ABB RobotStudio station: Project4.rsstnx

Station Project4 (saved by RobotStudio 23.2.10395.0)
Controller IRB140_6_81
  mechanical unit ROB_1: IRB140_6_81_C_03, 6 joints, base frame (0, 0, 0) mm
Layout (positions relative to the parent item):
  - IRB140_6_81_C_03 [mechanism, from %ABB.RobotStudio.Models.IRB140%\IRB140_6_81_C_G_03.rslib] at (0, 0, 0) mm; joint values [0.7528, 0.4246, 0.2198, -0.8632, 0.587, 1.4078] (rad or m)
  - Cubo_2 [part] at (500, 400, 0) mm, rotated rx 90 ry 0 rz 0 deg, size 180 x 200 x 180 mm
  - MyNewTool [mechanism] at (421.04, 356.95, 400.53) mm, rotated rx 180 ry 38 rz 180 deg
      TCP CualquierCosa at (131.19, 0, 127.78) mm, rotated rx 0 ry 75 rz 0 deg
      links: BaseMarcador
  - MyTool [mechanism, from Training Objects\myTool.rslib] at (421.04, 356.95, 400.53) mm, rotated rx 180 ry 38 rz 180 deg
Attachment: MyNewTool is attached to IRB140_6_81_C_03 / Link6
Attachment: MyTool is attached to IRB140_6_81_C_03 / Link6
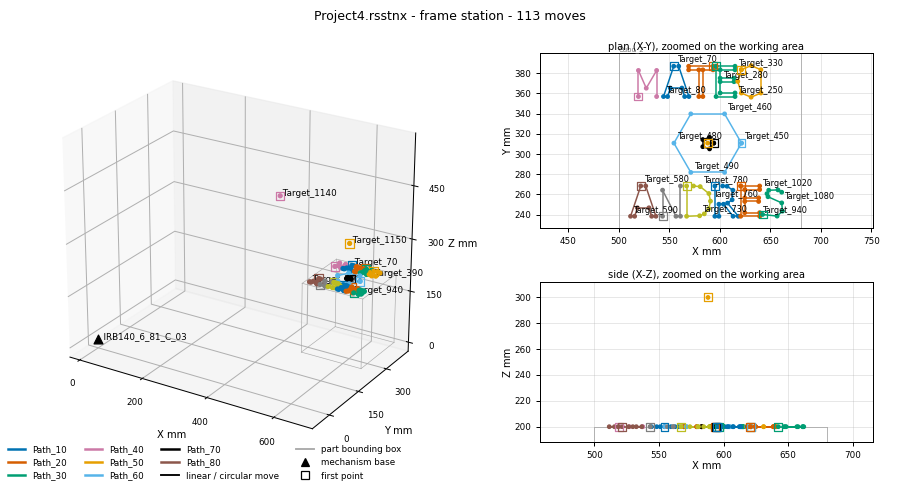
[picture p0: tool path of Project4.rsstnx in frame station, 113 of 113 moves have a stored position in this frame; points joined in program order, loops and branches not executed]
Targets, tools, work objects and paths stored in the station, written as RAPID:
! task T_ROB1
MODULE Module1
  PERS wobjdata Workobject_8:=[FALSE,TRUE,"",[[150,100,0],[1,0,0,0]],[[351.920963746,301.866615458,180],[0,0.710877818,0.703315525,0]]];
  CONST robtarget Target_10:=[[-44.732003119,17.911406594,-20],[0.703315525,0,0,-0.710877818],[0,0,0,0],[9E+09,9E+09,9E+09,9E+09,9E+09,9E+09]];
  CONST robtarget Target_20:=[[-18.89069334,17.635029753,-20],[0.703315525,0,0,-0.710877818],[0,0,0,0],[9E+09,9E+09,9E+09,9E+09,9E+09,9E+09]];
  CONST robtarget Target_30:=[[-36.383734505,25.577831517,-20],[0.703315525,0,0,-0.710877818],[0,0,0,0],[9E+09,9E+09,9E+09,9E+09,9E+09,9E+09]];
  CONST robtarget Target_40:=[[-18.698035542,35.64858624,-20],[0.703315525,0,0,-0.710877818],[0,0,0,0],[9E+09,9E+09,9E+09,9E+09,9E+09,9E+09]];
  CONST robtarget Target_50:=[[-44.539345321,35.924963081,-20],[0.703315525,0,0,-0.710877818],[0,0,0,0],[9E+09,9E+09,9E+09,9E+09,9E+09,9E+09]];
  CONST robtarget Target_60:=[[-14.355335815,52.933587211,-20],[0.703315525,0,0,-0.710877818],[0,0,0,0],[9E+09,9E+09,9E+09,9E+09,9E+09,9E+09]];
  CONST robtarget Target_70:=[[-14.359843041,52.548052351,-20],[0.703315525,0,0,-0.710877818],[0,0,0,0],[9E+09,9E+09,9E+09,9E+09,9E+09,9E+09]];
  CONST robtarget Target_80:=[[-44.466286156,42.756014866,-20],[0.703315525,0,0,-0.710877818],[0,0,0,0],[9E+09,9E+09,9E+09,9E+09,9E+09,9E+09]];
  CONST robtarget Target_90:=[[-44.423126649,46.791440476,-20],[0.703315525,0,0,-0.710877818],[0,0,0,0],[9E+09,9E+09,9E+09,9E+09,9E+09,9E+09]];
  CONST robtarget Target_100:=[[-36.007128456,49.424438298,-20],[0.703315525,0,0,-0.710877818],[0,0,0,0],[9E+09,9E+09,9E+09,9E+09,9E+09,9E+09]];
  CONST robtarget Target_110:=[[-35.884669856,60.874350721,-20],[0.703315525,0,0,-0.710877818],[0,0,0,0],[9E+09,9E+09,9E+09,9E+09,9E+09,9E+09]];
  CONST robtarget Target_120:=[[-44.242428715,63.686746492,-20],[0.703315525,0,0,-0.710877818],[0,0,0,0],[9E+09,9E+09,9E+09,9E+09,9E+09,9E+09]];
  CONST robtarget Target_130:=[[-44.197449229,67.892340652,-20],[0.703315525,0,0,-0.710877818],[0,0,0,0],[9E+09,9E+09,9E+09,9E+09,9E+09,9E+09]];
  CONST robtarget Target_140:=[[-14.307323641,57.458630502,-20],[0.703315525,0,0,-0.710877818],[0,0,0,0],[9E+09,9E+09,9E+09,9E+09,9E+09,9E+09]];
  CONST robtarget Target_150:=[[-13.943587799,91.468030671,-20],[0.703315525,0,0,-0.710877818],[0,0,0,0],[9E+09,9E+09,9E+09,9E+09,9E+09,9E+09]];
  CONST robtarget Target_160:=[[-14.201504851,67.352716184,-20],[0.703315525,0,0,-0.710877818],[0,0,0,0],[9E+09,9E+09,9E+09,9E+09,9E+09,9E+09]];
  CONST robtarget Target_170:=[[-17.750734604,67.39067575,-20],[0.703315525,0,0,-0.710877818],[0,0,0,0],[9E+09,9E+09,9E+09,9E+09,9E+09,9E+09]];
  CONST robtarget Target_180:=[[-17.643095834,77.454929981,-20],[0.703315525,0,0,-0.710877818],[0,0,0,0],[9E+09,9E+09,9E+09,9E+09,9E+09,9E+09]];
  CONST robtarget Target_190:=[[-44.092150433,77.737806747,-20],[0.703315525,0,0,-0.710877818],[0,0,0,0],[9E+09,9E+09,9E+09,9E+09,9E+09,9E+09]];
  CONST robtarget Target_200:=[[-44.04951092,81.724612772,-20],[0.703315525,0,0,-0.710877818],[0,0,0,0],[9E+09,9E+09,9E+09,9E+09,9E+09,9E+09]];
  CONST robtarget Target_210:=[[-17.600456321,81.441736005,-20],[0.703315525,0,0,-0.710877818],[0,0,0,0],[9E+09,9E+09,9E+09,9E+09,9E+09,9E+09]];
  CONST robtarget Target_220:=[[-17.492817552,91.505990237,-20],[0.703315525,0,0,-0.710877818],[0,0,0,0],[9E+09,9E+09,9E+09,9E+09,9E+09,9E+09]];
  CONST robtarget Target_230:=[[-13.91108817,94.506754775,-20],[0.703315525,0,0,-0.710877818],[0,0,0,0],[9E+09,9E+09,9E+09,9E+09,9E+09,9E+09]];
  CONST robtarget Target_240:=[[-43.909372522,94.827591107,-20],[0.703315525,0,0,-0.710877818],[0,0,0,0],[9E+09,9E+09,9E+09,9E+09,9E+09,9E+09]];
  CONST robtarget Target_250:=[[-43.708654816,113.594751171,-20],[0.703315525,0,0,-0.710877818],[0,0,0,0],[9E+09,9E+09,9E+09,9E+09,9E+09,9E+09]];
  CONST robtarget Target_260:=[[-40.159425063,113.556791605,-20],[0.703315525,0,0,-0.710877818],[0,0,0,0],[9E+09,9E+09,9E+09,9E+09,9E+09,9E+09]];
  CONST robtarget Target_270:=[[-40.317503256,98.776437565,-20],[0.703315525,0,0,-0.710877818],[0,0,0,0],[9E+09,9E+09,9E+09,9E+09,9E+09,9E+09]];
  CONST robtarget Target_280:=[[-29.18361814,98.657358926,-20],[0.703315525,0,0,-0.710877818],[0,0,0,0],[9E+09,9E+09,9E+09,9E+09,9E+09,9E+09]];
  CONST robtarget Target_290:=[[-29.036199825,112.44101146,-20],[0.703315525,0,0,-0.710877818],[0,0,0,0],[9E+09,9E+09,9E+09,9E+09,9E+09,9E+09]];
  CONST robtarget Target_300:=[[-25.486970072,112.403051894,-20],[0.703315525,0,0,-0.710877818],[0,0,0,0],[9E+09,9E+09,9E+09,9E+09,9E+09,9E+09]];
  CONST robtarget Target_310:=[[-25.634388387,98.61939936,-20],[0.703315525,0,0,-0.710877818],[0,0,0,0],[9E+09,9E+09,9E+09,9E+09,9E+09,9E+09]];
  CONST robtarget Target_320:=[[-17.417678411,98.531520364,-20],[0.703315525,0,0,-0.710877818],[0,0,0,0],[9E+09,9E+09,9E+09,9E+09,9E+09,9E+09]];
  CONST robtarget Target_330:=[[-17.259600218,113.311874405,-20],[0.703315525,0,0,-0.710877818],[0,0,0,0],[9E+09,9E+09,9E+09,9E+09,9E+09,9E+09]];
  CONST robtarget Target_340:=[[-13.710370465,113.273914839,-20],[0.703315525,0,0,-0.710877818],[0,0,0,0],[9E+09,9E+09,9E+09,9E+09,9E+09,9E+09]];
  CONST robtarget Target_350:=[[-13.91108817,94.506754775,-20],[0.703315525,0,0,-0.710877818],[0,0,0,0],[9E+09,9E+09,9E+09,9E+09,9E+09,9E+09]];
  CONST robtarget Target_360:=[[-17.07097202,119.58250097,-20],[0.703315525,0,0,-0.710877818],[0,0,0,0],[9E+09,9E+09,9E+09,9E+09,9E+09,9E+09]];
  CONST robtarget Target_370:=[[-28.680912967,116.108410216,-20],[0.703315525,0,0,-0.710877818],[0,0,0,0],[9E+09,9E+09,9E+09,9E+09,9E+09,9E+09]];
  CONST robtarget Target_380:=[[-40.189844998,119.805448351,-20],[0.703315525,0,0,-0.710877818],[0,0,0,0],[9E+09,9E+09,9E+09,9E+09,9E+09,9E+09]];
  CONST robtarget Target_390:=[[-44.170411377,129.524425398,-20],[0.703315525,0,0,-0.710877818],[0,0,0,0],[9E+09,9E+09,9E+09,9E+09,9E+09,9E+09]];
  CONST robtarget Target_400:=[[-39.982887363,139.156043443,-20],[0.703315525,0,0,-0.710877818],[0,0,0,0],[9E+09,9E+09,9E+09,9E+09,9E+09,9E+09]];
  CONST robtarget Target_410:=[[-28.39725621,142.630394193,-20],[0.703315525,0,0,-0.710877818],[0,0,0,0],[9E+09,9E+09,9E+09,9E+09,9E+09,9E+09]];
  CONST robtarget Target_420:=[[-16.864274383,138.908786269,-20],[0.703315525,0,0,-0.710877818],[0,0,0,0],[9E+09,9E+09,9E+09,9E+09,9E+09,9E+09]];
  CONST robtarget Target_430:=[[-12.908017797,129.19006922,-20],[0.703315525,0,0,-0.710877818],[0,0,0,0],[9E+09,9E+09,9E+09,9E+09,9E+09,9E+09]];
  CONST robtarget Target_440:=[[-17.07097202,119.58250097,-20],[0.703315525,0,0,-0.710877818],[0,0,0,0],[9E+09,9E+09,9E+09,9E+09,9E+09,9E+09]];
  CONST robtarget Target_450:=[[-89.795859571,120.450633168,-20],[0.703315525,0,0,-0.710877818],[0,0,0,0],[9E+09,9E+09,9E+09,9E+09,9E+09,9E+09]];
  CONST robtarget Target_460:=[[-61.00596514,103.415679147,-20],[0.703315525,0,0,-0.710877818],[0,0,0,0],[9E+09,9E+09,9E+09,9E+09,9E+09,9E+09]];
  CONST robtarget Target_470:=[[-61.363720858,69.965422187,-20],[0.703315525,0,0,-0.710877818],[0,0,0,0],[9E+09,9E+09,9E+09,9E+09,9E+09,9E+09]];
  CONST robtarget Target_480:=[[-90.511371008,53.550119248,-20],[0.703315525,0,0,-0.710877818],[0,0,0,0],[9E+09,9E+09,9E+09,9E+09,9E+09,9E+09]];
  CONST robtarget Target_490:=[[-119.30126544,70.585073268,-20],[0.703315525,0,0,-0.710877818],[0,0,0,0],[9E+09,9E+09,9E+09,9E+09,9E+09,9E+09]];
  CONST robtarget Target_500:=[[-118.943509722,104.035330228,-20],[0.703315525,0,0,-0.710877818],[0,0,0,0],[9E+09,9E+09,9E+09,9E+09,9E+09,9E+09]];
  CONST robtarget Target_510:=[[-89.795859571,120.450633168,-20],[0.703315525,0,0,-0.710877818],[0,0,0,0],[9E+09,9E+09,9E+09,9E+09,9E+09,9E+09]];
  CONST robtarget Target_520:=[[-90.089448023,93.000033078,-20],[0.703315525,0,0,-0.710877818],[0,0,0,0],[9E+09,9E+09,9E+09,9E+09,9E+09,9E+09]];
  CONST robtarget Target_530:=[[-95.839799276,88.915398838,-20],[0.703315525,0,0,-0.710877818],[0,0,0,0],[9E+09,9E+09,9E+09,9E+09,9E+09,9E+09]];
  CONST robtarget Target_540:=[[-93.732037526,82.184268413,-20],[0.703315525,0,0,-0.710877818],[0,0,0,0],[9E+09,9E+09,9E+09,9E+09,9E+09,9E+09]];
  CONST robtarget Target_550:=[[-86.679017871,82.108835267,-20],[0.703315525,0,0,-0.710877818],[0,0,0,0],[9E+09,9E+09,9E+09,9E+09,9E+09,9E+09]];
  CONST robtarget Target_560:=[[-84.427773752,88.793345444,-20],[0.703315525,0,0,-0.710877818],[0,0,0,0],[9E+09,9E+09,9E+09,9E+09,9E+09,9E+09]];
  CONST robtarget Target_570:=[[-90.089448023,93.000033078,-20],[0.703315525,0,0,-0.710877818],[0,0,0,0],[9E+09,9E+09,9E+09,9E+09,9E+09,9E+09]];
  CONST robtarget Target_580:=[[-133.307718567,21.169891203,-20],[0.703315525,0,0,-0.710877818],[0,0,0,0],[9E+09,9E+09,9E+09,9E+09,9E+09,9E+09]];
  CONST robtarget Target_590:=[[-163.414161682,11.377853719,-20],[0.703315525,0,0,-0.710877818],[0,0,0,0],[9E+09,9E+09,9E+09,9E+09,9E+09,9E+09]];
  CONST robtarget Target_600:=[[-163.371002175,15.413279329,-20],[0.703315525,0,0,-0.710877818],[0,0,0,0],[9E+09,9E+09,9E+09,9E+09,9E+09,9E+09]];
  CONST robtarget Target_610:=[[-154.955003982,18.046277151,-20],[0.703315525,0,0,-0.710877818],[0,0,0,0],[9E+09,9E+09,9E+09,9E+09,9E+09,9E+09]];
  CONST robtarget Target_620:=[[-154.832545382,29.496189573,-20],[0.703315525,0,0,-0.710877818],[0,0,0,0],[9E+09,9E+09,9E+09,9E+09,9E+09,9E+09]];
  CONST robtarget Target_630:=[[-163.190304241,32.308585345,-20],[0.703315525,0,0,-0.710877818],[0,0,0,0],[9E+09,9E+09,9E+09,9E+09,9E+09,9E+09]];
  CONST robtarget Target_640:=[[-163.145324755,36.514179505,-20],[0.703315525,0,0,-0.710877818],[0,0,0,0],[9E+09,9E+09,9E+09,9E+09,9E+09,9E+09]];
  CONST robtarget Target_650:=[[-133.255199167,26.080469355,-20],[0.703315525,0,0,-0.710877818],[0,0,0,0],[9E+09,9E+09,9E+09,9E+09,9E+09,9E+09]];
  CONST robtarget Target_660:=[[-163.075125558,43.077823569,-20],[0.703315525,0,0,-0.710877818],[0,0,0,0],[9E+09,9E+09,9E+09,9E+09,9E+09,9E+09]];
  CONST robtarget Target_670:=[[-137.209505986,42.801186731,-20],[0.703315525,0,0,-0.710877818],[0,0,0,0],[9E+09,9E+09,9E+09,9E+09,9E+09,9E+09]];
  CONST robtarget Target_680:=[[-162.93316718,56.350970454,-20],[0.703315525,0,0,-0.710877818],[0,0,0,0],[9E+09,9E+09,9E+09,9E+09,9E+09,9E+09]];
  CONST robtarget Target_690:=[[-162.885327727,60.823972334,-20],[0.703315525,0,0,-0.710877818],[0,0,0,0],[9E+09,9E+09,9E+09,9E+09,9E+09,9E+09]];
  CONST robtarget Target_700:=[[-132.887043375,60.503136001,-20],[0.703315525,0,0,-0.710877818],[0,0,0,0],[9E+09,9E+09,9E+09,9E+09,9E+09,9E+09]];
  CONST robtarget Target_710:=[[-132.822044118,66.580584209,-20],[0.703315525,0,0,-0.710877818],[0,0,0,0],[9E+09,9E+09,9E+09,9E+09,9E+09,9E+09]];
  CONST robtarget Target_720:=[[-162.82032847,66.901420541,-20],[0.703315525,0,0,-0.710877818],[0,0,0,0],[9E+09,9E+09,9E+09,9E+09,9E+09,9E+09]];
  CONST robtarget Target_730:=[[-162.19620419,79.792565697,-20],[0.703315525,0,0,-0.710877818],[0,0,0,0],[9E+09,9E+09,9E+09,9E+09,9E+09,9E+09]];
  CONST robtarget Target_740:=[[-160.226201123,84.403041466,-20],[0.703315525,0,0,-0.710877818],[0,0,0,0],[9E+09,9E+09,9E+09,9E+09,9E+09,9E+09]];
  CONST robtarget Target_750:=[[-155.024815588,88.80876908,-20],[0.703315525,0,0,-0.710877818],[0,0,0,0],[9E+09,9E+09,9E+09,9E+09,9E+09,9E+09]];
  CONST robtarget Target_760:=[[-147.592518979,90.394690796,-20],[0.703315525,0,0,-0.710877818],[0,0,0,0],[9E+09,9E+09,9E+09,9E+09,9E+09,9E+09]];
  CONST robtarget Target_770:=[[-140.061358111,88.721670288,-20],[0.703315525,0,0,-0.710877818],[0,0,0,0],[9E+09,9E+09,9E+09,9E+09,9E+09,9E+09]];
  CONST robtarget Target_780:=[[-133.310060379,80.054969359,-20],[0.703315525,0,0,-0.710877818],[0,0,0,0],[9E+09,9E+09,9E+09,9E+09,9E+09,9E+09]];
  CONST robtarget Target_790:=[[-132.748984953,73.411635994,-20],[0.703315525,0,0,-0.710877818],[0,0,0,0],[9E+09,9E+09,9E+09,9E+09,9E+09,9E+09]];
  CONST robtarget Target_800:=[[-132.522787539,94.561155755,-20],[0.703315525,0,0,-0.710877818],[0,0,0,0],[9E+09,9E+09,9E+09,9E+09,9E+09,9E+09]];
  CONST robtarget Target_810:=[[-162.521071891,94.881992088,-20],[0.703315525,0,0,-0.710877818],[0,0,0,0],[9E+09,9E+09,9E+09,9E+09,9E+09,9E+09]];
  CONST robtarget Target_820:=[[-162.478432378,98.868798112,-20],[0.703315525,0,0,-0.710877818],[0,0,0,0],[9E+09,9E+09,9E+09,9E+09,9E+09,9E+09]];
  CONST robtarget Target_830:=[[-150.542324099,98.741139572,-20],[0.703315525,0,0,-0.710877818],[0,0,0,0],[9E+09,9E+09,9E+09,9E+09,9E+09,9E+09]];
  CONST robtarget Target_840:=[[-150.493444657,103.311380624,-20],[0.703315525,0,0,-0.710877818],[0,0,0,0],[9E+09,9E+09,9E+09,9E+09,9E+09,9E+09]];
  CONST robtarget Target_850:=[[-162.328154096,112.919858368,-20],[0.703315525,0,0,-0.710877818],[0,0,0,0],[9E+09,9E+09,9E+09,9E+09,9E+09,9E+09]];
  CONST robtarget Target_860:=[[-162.272774729,118.097844241,-20],[0.703315525,0,0,-0.710877818],[0,0,0,0],[9E+09,9E+09,9E+09,9E+09,9E+09,9E+09]];
  CONST robtarget Target_870:=[[-149.332554674,107.286226785,-20],[0.703315525,0,0,-0.710877818],[0,0,0,0],[9E+09,9E+09,9E+09,9E+09,9E+09,9E+09]];
  CONST robtarget Target_880:=[[-145.989958302,111.796928447,-20],[0.703315525,0,0,-0.710877818],[0,0,0,0],[9E+09,9E+09,9E+09,9E+09,9E+09,9E+09]];
  CONST robtarget Target_890:=[[-136.525258985,112.461548077,-20],[0.703315525,0,0,-0.710877818],[0,0,0,0],[9E+09,9E+09,9E+09,9E+09,9E+09,9E+09]];
  CONST robtarget Target_900:=[[-132.673521629,106.609648068,-20],[0.703315525,0,0,-0.710877818],[0,0,0,0],[9E+09,9E+09,9E+09,9E+09,9E+09,9E+09]];
  CONST robtarget Target_910:=[[-132.440108484,102.291669875,-20],[0.703315525,0,0,-0.710877818],[0,0,0,0],[9E+09,9E+09,9E+09,9E+09,9E+09,9E+09]];
  CONST robtarget Target_920:=[[-132.249010668,120.159367605,-20],[0.703315525,0,0,-0.710877818],[0,0,0,0],[9E+09,9E+09,9E+09,9E+09,9E+09,9E+09]];
  CONST robtarget Target_930:=[[-162.24729502,120.480203938,-20],[0.703315525,0,0,-0.710877818],[0,0,0,0],[9E+09,9E+09,9E+09,9E+09,9E+09,9E+09]];
  CONST robtarget Target_940:=[[-162.046577315,139.247364003,-20],[0.703315525,0,0,-0.710877818],[0,0,0,0],[9E+09,9E+09,9E+09,9E+09,9E+09,9E+09]];
  CONST robtarget Target_950:=[[-158.497347562,139.209404437,-20],[0.703315525,0,0,-0.710877818],[0,0,0,0],[9E+09,9E+09,9E+09,9E+09,9E+09,9E+09]];
  CONST robtarget Target_960:=[[-158.655425755,124.429050396,-20],[0.703315525,0,0,-0.710877818],[0,0,0,0],[9E+09,9E+09,9E+09,9E+09,9E+09,9E+09]];
  CONST robtarget Target_970:=[[-147.521540639,124.309971757,-20],[0.703315525,0,0,-0.710877818],[0,0,0,0],[9E+09,9E+09,9E+09,9E+09,9E+09,9E+09]];
  CONST robtarget Target_980:=[[-147.374122324,138.093624292,-20],[0.703315525,0,0,-0.710877818],[0,0,0,0],[9E+09,9E+09,9E+09,9E+09,9E+09,9E+09]];
  CONST robtarget Target_990:=[[-143.824892571,138.055664726,-20],[0.703315525,0,0,-0.710877818],[0,0,0,0],[9E+09,9E+09,9E+09,9E+09,9E+09,9E+09]];
  CONST robtarget Target_1000:=[[-143.972310886,124.272012191,-20],[0.703315525,0,0,-0.710877818],[0,0,0,0],[9E+09,9E+09,9E+09,9E+09,9E+09,9E+09]];
  CONST robtarget Target_1010:=[[-135.755600909,124.184133196,-20],[0.703315525,0,0,-0.710877818],[0,0,0,0],[9E+09,9E+09,9E+09,9E+09,9E+09,9E+09]];
  CONST robtarget Target_1020:=[[-135.597522716,138.964487236,-20],[0.703315525,0,0,-0.710877818],[0,0,0,0],[9E+09,9E+09,9E+09,9E+09,9E+09,9E+09]];
  CONST robtarget Target_1030:=[[-132.048292963,138.92652767,-20],[0.703315525,0,0,-0.710877818],[0,0,0,0],[9E+09,9E+09,9E+09,9E+09,9E+09,9E+09]];
  CONST robtarget Target_1040:=[[-132.249010668,120.159367605,-20],[0.703315525,0,0,-0.710877818],[0,0,0,0],[9E+09,9E+09,9E+09,9E+09,9E+09,9E+09]];
  CONST robtarget Target_1050:=[[-160.216712999,142.120989569,-20],[0.703315525,0,0,-0.710877818],[0,0,0,0],[9E+09,9E+09,9E+09,9E+09,9E+09,9E+09]];
  CONST robtarget Target_1060:=[[-161.691290881,156.554116518,-20],[0.703315525,0,0,-0.710877818],[0,0,0,0],[9E+09,9E+09,9E+09,9E+09,9E+09,9E+09]];
  CONST robtarget Target_1070:=[[-156.724423373,161.764667266,-20],[0.703315525,0,0,-0.710877818],[0,0,0,0],[9E+09,9E+09,9E+09,9E+09,9E+09,9E+09]];
  CONST robtarget Target_1080:=[[-148.551847998,160.960039377,-20],[0.703315525,0,0,-0.710877818],[0,0,0,0],[9E+09,9E+09,9E+09,9E+09,9E+09,9E+09]];
  CONST robtarget Target_1090:=[[-142.619608131,147.318020825,-20],[0.703315525,0,0,-0.710877818],[0,0,0,0],[9E+09,9E+09,9E+09,9E+09,9E+09,9E+09]];
  CONST robtarget Target_1100:=[[-139.6038288,146.276794793,-20],[0.703315525,0,0,-0.710877818],[0,0,0,0],[9E+09,9E+09,9E+09,9E+09,9E+09,9E+09]];
  CONST robtarget Target_1110:=[[-136.169973116,147.954105604,-20],[0.703315525,0,0,-0.710877818],[0,0,0,0],[9E+09,9E+09,9E+09,9E+09,9E+09,9E+09]];
  CONST robtarget Target_1120:=[[-135.743642036,157.127542438,-20],[0.703315525,0,0,-0.710877818],[0,0,0,0],[9E+09,9E+09,9E+09,9E+09,9E+09,9E+09]];
  CONST robtarget Target_1130:=[[-137.989503011,160.822760876,-20],[0.703315525,0,0,-0.710877818],[0,0,0,0],[9E+09,9E+09,9E+09,9E+09,9E+09,9E+09]];
  PERS tooldata CualquierCosa:=[TRUE,[[131.189,0,127.783],[0.79335334,0,0.608761429,0]],[1,[0,0,1],[1,0,0,0],0,0,0]];
  CONST robtarget Target_1140:=[[-463.655972586,103.338535401,-388.928],[0.703315525,0,0,-0.710877818],[0,0,0,0],[9E+09,9E+09,9E+09,9E+09,9E+09,9E+09]];
  CONST robtarget Target_1150:=[[-90.15334409,87.000160586,-120],[0.703315525,0,0,-0.710877818],[0,0,0,0],[9E+09,9E+09,9E+09,9E+09,9E+09,9E+09]];
  PERS tooldata MyTool:=[TRUE,[[31.792631019,0,229.638935148],[0.945518576,0,0.325568154,0]],[1,[0,0,1],[1,0,0,0],0,0,0]];
  PROC Path_10()
    MoveL Target_70,v1000,z100,CualquierCosa\WObj:=Workobject_8;
    MoveL Target_80,v1000,z100,CualquierCosa\WObj:=Workobject_8;
    MoveL Target_90,v1000,z100,CualquierCosa\WObj:=Workobject_8;
    MoveL Target_100,v1000,z100,CualquierCosa\WObj:=Workobject_8;
    MoveL Target_110,v1000,z100,CualquierCosa\WObj:=Workobject_8;
    MoveL Target_120,v1000,z100,CualquierCosa\WObj:=Workobject_8;
    MoveL Target_130,v1000,z100,CualquierCosa\WObj:=Workobject_8;
    MoveL Target_140,v1000,z100,CualquierCosa\WObj:=Workobject_8;
  ENDPROC
  PROC Path_20()
    MoveL Target_150,v1000,z100,CualquierCosa\WObj:=Workobject_8;
    MoveL Target_160,v1000,z100,CualquierCosa\WObj:=Workobject_8;
    MoveL Target_170,v1000,z100,CualquierCosa\WObj:=Workobject_8;
    MoveL Target_180,v1000,z100,CualquierCosa\WObj:=Workobject_8;
    MoveL Target_190,v1000,z100,CualquierCosa\WObj:=Workobject_8;
    MoveL Target_200,v1000,z100,CualquierCosa\WObj:=Workobject_8;
    MoveL Target_210,v1000,z100,CualquierCosa\WObj:=Workobject_8;
    MoveL Target_220,v1000,z100,CualquierCosa\WObj:=Workobject_8;
  ENDPROC
  LOCAL PROC Path_30()
    MoveL Target_230,v1000,z100,CualquierCosa\WObj:=Workobject_8;
    MoveL Target_240,v1000,z100,CualquierCosa\WObj:=Workobject_8;
    MoveL Target_250,v1000,z100,CualquierCosa\WObj:=Workobject_8;
    MoveL Target_260,v1000,z100,CualquierCosa\WObj:=Workobject_8;
    MoveL Target_270,v1000,z100,CualquierCosa\WObj:=Workobject_8;
    MoveL Target_280,v1000,z100,CualquierCosa\WObj:=Workobject_8;
    MoveL Target_290,v1000,z100,CualquierCosa\WObj:=Workobject_8;
    MoveL Target_300,v1000,z100,CualquierCosa\WObj:=Workobject_8;
    MoveL Target_310,v1000,z100,CualquierCosa\WObj:=Workobject_8;
    MoveL Target_320,v1000,z100,CualquierCosa\WObj:=Workobject_8;
    MoveL Target_330,v1000,z100,CualquierCosa\WObj:=Workobject_8;
    MoveL Target_340,v1000,z100,CualquierCosa\WObj:=Workobject_8;
    MoveL Target_350,v1000,z100,CualquierCosa\WObj:=Workobject_8;
  ENDPROC
  PROC Path_40()
    MoveL Target_10,v1000,z100,CualquierCosa\WObj:=Workobject_8;
    MoveL Target_20,v1000,z100,CualquierCosa\WObj:=Workobject_8;
    MoveL Target_30,v1000,z100,CualquierCosa\WObj:=Workobject_8;
    MoveL Target_40,v1000,z100,CualquierCosa\WObj:=Workobject_8;
    MoveL Target_50,v1000,z100,CualquierCosa\WObj:=Workobject_8;
  ENDPROC
  PROC main()
    Path_40;
  ENDPROC
  PROC Path_50()
    MoveL Target_360,v1000,z100,CualquierCosa\WObj:=Workobject_8;
    MoveL Target_370,v1000,z100,CualquierCosa\WObj:=Workobject_8;
    MoveL Target_380,v1000,z100,CualquierCosa\WObj:=Workobject_8;
    MoveL Target_390,v1000,z100,CualquierCosa\WObj:=Workobject_8;
    MoveL Target_400,v1000,z100,CualquierCosa\WObj:=Workobject_8;
    MoveL Target_420,v1000,z100,CualquierCosa\WObj:=Workobject_8;
    MoveL Target_430,v1000,z100,CualquierCosa\WObj:=Workobject_8;
    MoveL Target_440,v1000,z100,CualquierCosa\WObj:=Workobject_8;
  ENDPROC
  PROC Path_60()
    MoveL Target_450,v1000,z100,CualquierCosa\WObj:=Workobject_8;
    MoveL Target_460,v1000,z100,CualquierCosa\WObj:=Workobject_8;
    MoveL Target_470,v1000,z100,CualquierCosa\WObj:=Workobject_8;
    MoveL Target_480,v1000,z100,CualquierCosa\WObj:=Workobject_8;
    MoveL Target_490,v1000,z100,CualquierCosa\WObj:=Workobject_8;
    MoveL Target_500,v1000,z100,CualquierCosa\WObj:=Workobject_8;
    MoveL Target_510,v1000,z100,CualquierCosa\WObj:=Workobject_8;
  ENDPROC
  PROC Path_70()
    MoveL Target_520,v1000,z100,CualquierCosa\WObj:=Workobject_8;
    MoveL Target_530,v1000,z100,CualquierCosa\WObj:=Workobject_8;
    MoveL Target_540,v1000,z100,CualquierCosa\WObj:=Workobject_8;
    MoveL Target_550,v1000,z100,CualquierCosa\WObj:=Workobject_8;
    MoveL Target_560,v1000,z100,CualquierCosa\WObj:=Workobject_8;
    MoveL Target_570,v1000,z100,CualquierCosa\WObj:=Workobject_8;
  ENDPROC
  PROC Path_80()
    MoveL Target_580,v1000,z100,CualquierCosa\WObj:=Workobject_8;
    MoveL Target_590,v1000,z100,CualquierCosa\WObj:=Workobject_8;
    MoveL Target_600,v1000,z100,CualquierCosa\WObj:=Workobject_8;
    MoveL Target_610,v1000,z100,CualquierCosa\WObj:=Workobject_8;
    MoveL Target_620,v1000,z100,CualquierCosa\WObj:=Workobject_8;
    MoveL Target_630,v1000,z100,CualquierCosa\WObj:=Workobject_8;
    MoveL Target_640,v1000,z100,CualquierCosa\WObj:=Workobject_8;
    MoveL Target_650,v1000,z100,CualquierCosa\WObj:=Workobject_8;
  ENDPROC
  PROC Path_90()
    MoveL Target_660,v1000,z100,CualquierCosa\WObj:=Workobject_8;
    MoveL Target_670,v1000,z100,CualquierCosa\WObj:=Workobject_8;
    MoveL Target_680,v1000,z100,CualquierCosa\WObj:=Workobject_8;
    MoveL Target_690,v1000,z100,CualquierCosa\WObj:=Workobject_8;
    MoveL Target_700,v1000,z100,CualquierCosa\WObj:=Workobject_8;
  ENDPROC
  PROC Path_100()
    MoveL Target_710,v1000,z100,CualquierCosa\WObj:=Workobject_8;
    MoveL Target_720,v1000,z100,CualquierCosa\WObj:=Workobject_8;
    MoveL Target_730,v1000,z100,CualquierCosa\WObj:=Workobject_8;
    MoveL Target_740,v1000,z100,CualquierCosa\WObj:=Workobject_8;
    MoveL Target_750,v1000,z100,CualquierCosa\WObj:=Workobject_8;
    MoveL Target_760,v1000,z100,CualquierCosa\WObj:=Workobject_8;
    MoveL Target_770,v1000,z100,CualquierCosa\WObj:=Workobject_8;
    MoveL Target_780,v1000,z100,CualquierCosa\WObj:=Workobject_8;
    MoveL Target_790,v1000,z100,CualquierCosa\WObj:=Workobject_8;
  ENDPROC
  PROC Path_110()
    MoveL Target_800,v1000,z100,CualquierCosa\WObj:=Workobject_8;
    MoveL Target_810,v1000,z100,CualquierCosa\WObj:=Workobject_8;
    MoveL Target_820,v1000,z100,CualquierCosa\WObj:=Workobject_8;
    MoveL Target_830,v1000,z100,CualquierCosa\WObj:=Workobject_8;
    MoveL Target_840,v1000,z100,CualquierCosa\WObj:=Workobject_8;
    MoveL Target_850,v1000,z100,CualquierCosa\WObj:=Workobject_8;
    MoveL Target_860,v1000,z100,CualquierCosa\WObj:=Workobject_8;
    MoveL Target_870,v1000,z100,CualquierCosa\WObj:=Workobject_8;
    MoveL Target_880,v1000,z100,CualquierCosa\WObj:=Workobject_8;
    MoveL Target_890,v1000,z100,CualquierCosa\WObj:=Workobject_8;
    MoveL Target_900,v1000,z100,CualquierCosa\WObj:=Workobject_8;
    MoveL Target_910,v1000,z100,CualquierCosa\WObj:=Workobject_8;
  ENDPROC
  PROC Path_120()
    MoveL Target_920,v1000,z100,CualquierCosa\WObj:=Workobject_8;
    MoveL Target_930,v1000,z100,CualquierCosa\WObj:=Workobject_8;
    MoveL Target_940,v1000,z100,CualquierCosa\WObj:=Workobject_8;
    MoveL Target_950,v1000,z100,CualquierCosa\WObj:=Workobject_8;
    MoveL Target_960,v1000,z100,CualquierCosa\WObj:=Workobject_8;
    MoveL Target_970,v1000,z100,CualquierCosa\WObj:=Workobject_8;
    MoveL Target_980,v1000,z100,CualquierCosa\WObj:=Workobject_8;
    MoveL Target_990,v1000,z100,CualquierCosa\WObj:=Workobject_8;
    MoveL Target_1000,v1000,z100,CualquierCosa\WObj:=Workobject_8;
    MoveL Target_1010,v1000,z100,CualquierCosa\WObj:=Workobject_8;
    MoveL Target_1020,v1000,z100,CualquierCosa\WObj:=Workobject_8;
    MoveL Target_1030,v1000,z100,CualquierCosa\WObj:=Workobject_8;
    MoveL Target_1040,v1000,z100,CualquierCosa\WObj:=Workobject_8;
  ENDPROC
  PROC Path_130()
    MoveL Target_1050,v1000,z100,CualquierCosa\WObj:=Workobject_8;
    MoveL Target_1060,v1000,z100,CualquierCosa\WObj:=Workobject_8;
    MoveL Target_1070,v1000,z100,CualquierCosa\WObj:=Workobject_8;
    MoveL Target_1080,v1000,z100,CualquierCosa\WObj:=Workobject_8;
    MoveL Target_1090,v1000,z100,CualquierCosa\WObj:=Workobject_8;
    MoveL Target_1100,v1000,z100,CualquierCosa\WObj:=Workobject_8;
    MoveL Target_1110,v1000,z100,CualquierCosa\WObj:=Workobject_8;
    MoveL Target_1120,v1000,z100,CualquierCosa\WObj:=Workobject_8;
    MoveL Target_1130,v1000,z100,CualquierCosa\WObj:=Workobject_8;
  ENDPROC
  PROC home()
    MoveL Target_1140,v1000,z100,CualquierCosa\WObj:=Workobject_8;
  ENDPROC
  PROC home_2()
    MoveL Target_1150,v1000,z100,CualquierCosa\WObj:=Workobject_8;
  ENDPROC
ENDMODULE

